FUNCTION_BLOCK FB_SimulatedOutOpen_DG IMPLEMENTS ITF_Regelschuif_OutOpen_DG
VAR
	internalState : BOOL := FALSE;
END_VAR

METHOD set : BOOL
VAR_INPUT
	state : BOOL;
END_VAR
internalState := state;
END_METHOD

END_FUNCTION_BLOCK

(* stored: Version 1.1.0.1, ProductVersion 3.1.4026.8
   POU FB_SimulatedOutOpen_DG: Id {9d9c518a-3a46-4ca8-a5b8-2c0ac1be4c7b}, SpecialFunc None
   Method set: Id {bcd0bac6-3ed9-4947-a075-8f2420f81498} *)
